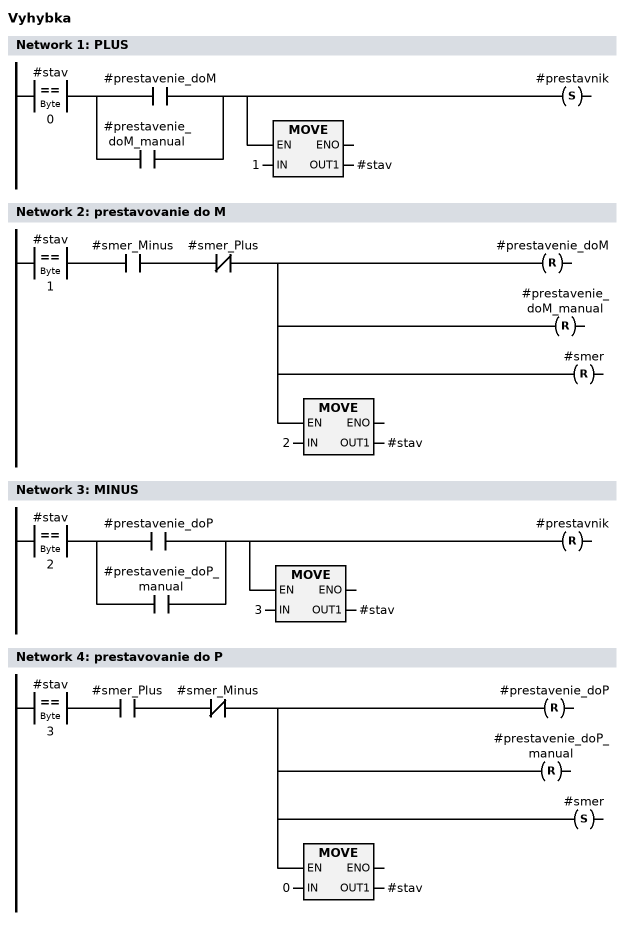
   RUNG wire#powerrail
      { S7_Templates := "SrcType := Byte" } EQ_Contact(in1 := #stav, in2 := 0)
      wire#w1
      Contact( #prestavenie_doM )
      wire#w2
      S_Coil( #prestavnik )
   END_RUNG
   RUNG wire#w1
      Contact( #prestavenie_doM_manual )
   END_RUNG wire#w2
   RUNG wire#w2
      Move(in := 1, out1 => #stav)
   END_RUNG
   // the same network as SCL:
   IF (#stav = 0) AND (#prestavenie_doM OR #prestavenie_doM_manual) THEN
       #prestavnik := TRUE;
       #stav := 1;
   END_IF;
END_REGION

REGION Network 2: prestavovanie do M
   RUNG wire#powerrail
      { S7_Templates := "SrcType := Byte" } EQ_Contact(in1 := #stav, in2 := 1)
      Contact( #smer_Minus )
      I_Contact( #smer_Plus )
      wire#w1
      R_Coil( #prestavenie_doM )
   END_RUNG
   RUNG wire#w1
      R_Coil( #prestavenie_doM_manual )
   END_RUNG
   RUNG wire#w1
      R_Coil( #smer )
   END_RUNG
   RUNG wire#w1
      Move(in := 2, out1 => #stav)
   END_RUNG
   // the same network as SCL:
   IF (#stav = 1) AND #smer_Minus AND NOT #smer_Plus THEN
       #prestavenie_doM := FALSE;
       #prestavenie_doM_manual := FALSE;
       #smer := FALSE;
       #stav := 2;
   END_IF;
END_REGION

REGION Network 3: MINUS
   RUNG wire#powerrail
      { S7_Templates := "SrcType := Byte" } EQ_Contact(in1 := #stav, in2 := 2)
      wire#w1
      Contact( #prestavenie_doP )
      wire#w2
      R_Coil( #prestavnik )
   END_RUNG
   RUNG wire#w1
      Contact( #prestavenie_doP_manual )
   END_RUNG wire#w2
   RUNG wire#w2
      Move(in := 3, out1 => #stav)
   END_RUNG
   // the same network as SCL:
   IF (#stav = 2) AND (#prestavenie_doP OR #prestavenie_doP_manual) THEN
       #prestavnik := FALSE;
       #stav := 3;
   END_IF;
END_REGION

REGION Network 4: prestavovanie do P
   RUNG wire#powerrail
      { S7_Templates := "SrcType := Byte" } EQ_Contact(in1 := #stav, in2 := 3)
      Contact( #smer_Plus )
      I_Contact( #smer_Minus )
      wire#w1
      R_Coil( #prestavenie_doP )
   END_RUNG
   RUNG wire#w1
      R_Coil( #prestavenie_doP_manual )
   END_RUNG
   RUNG wire#w1
      S_Coil( #smer )
   END_RUNG
   RUNG wire#w1
      Move(in := 0, out1 => #stav)
   END_RUNG
   // the same network as SCL:
   IF (#stav = 3) AND #smer_Plus AND NOT #smer_Minus THEN
       #prestavenie_doP := FALSE;
       #prestavenie_doP_manual := FALSE;
       #smer := TRUE;
       #stav := 0;
   END_IF;
END_REGION
END_FUNCTION_BLOCK

FUNCTION_BLOCK "Detekcia_Smeru_Jazdy"   // FB8, SCL
{ S7_Optimized_Access := 'TRUE' }
VERSION : 0.1
   VAR_INPUT
      PU_AB : Bool;   // Priblizovaci usek-smer AB
      AU : Bool;   // Anulovaci usek
      PU_BA : Bool;   // Priblizovaci usek-smer BA
   END_VAR
   VAR_OUTPUT
      S_AB : Bool;   // Smer A->B
      S_BA : Bool;   // Smer B->A
   END_VAR
   VAR
      Stav : USInt;
   END_VAR
BEGIN
   CASE #Stav OF
       0:
           #S_AB := FALSE;
           #S_BA := FALSE;

           IF ((#PU_AB) AND NOT (#AU) AND NOT (#PU_BA)) THEN
               #Stav := 1;
           END_IF;

           IF (NOT (#PU_AB) AND NOT (#AU) AND (#PU_BA)) THEN
               #Stav := 2;
           END_IF;

       1:
           #S_AB := TRUE;
           #S_BA := FALSE;

           IF (NOT (#PU_AB) AND NOT (#AU) AND NOT (#PU_BA)) THEN
               #Stav := 0;
           END_IF;

       2:
           #S_AB := FALSE;
           #S_BA := TRUE;

           IF (NOT (#PU_AB) AND NOT (#AU) AND NOT (#PU_BA)) THEN
               #Stav := 0;
           END_IF;
   END_CASE;
END_FUNCTION_BLOCK

ORGANIZATION_BLOCK "Main"   // OB1, LAD, ProgramCycle
TITLE = "Main Program Sweep (Cycle)"
{ S7_Optimized_Access := 'TRUE' }
VERSION : 0.1
   VAR_INPUT
      Initial_Call : Bool;   // Initial call of this OB
      Remanence : Bool;   // =True, if remanent data are available
   END_VAR
BEGIN

REGION Network 1: Lo/PrLo
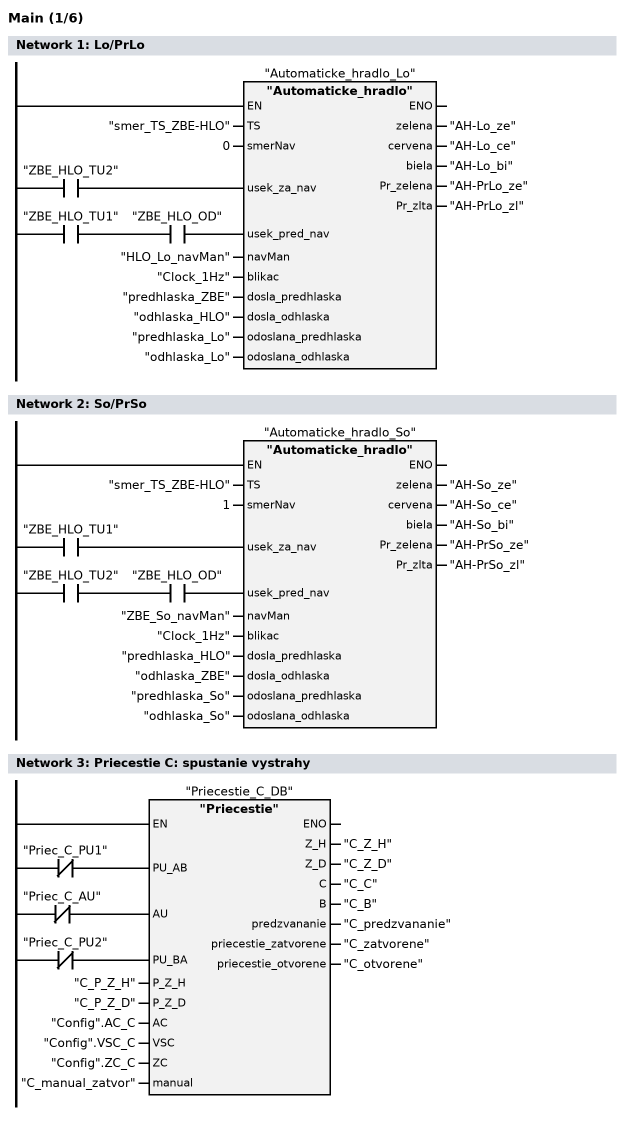
   RUNG wire#powerrail
      "Automaticke_hradlo_Lo"(usek_za_nav := wire#w1, usek_pred_nav := wire#w2, TS := "smer_TS_ZBE-HLO", smerNav := 0, navMan := "HLO_Lo_navMan", blikac := "Clock_1Hz", dosla_predhlaska := "predhlaska_ZBE", dosla_odhlaska := "odhlaska_HLO", odoslana_predhlaska := "predhlaska_Lo", odoslana_odhlaska := "odhlaska_Lo", zelena => "AH-Lo_ze", cervena => "AH-Lo_ce", biela => "AH-Lo_bi", Pr_zelena => "AH-PrLo_ze", Pr_zlta => "AH-PrLo_zl")
   END_RUNG
   RUNG wire#powerrail
      Contact( "ZBE_HLO_TU2" )
   END_RUNG wire#w1
   RUNG wire#powerrail
      Contact( "ZBE_HLO_TU1" )
      Contact( "ZBE_HLO_OD" )
   END_RUNG wire#w2
   // the same network as SCL:
   "Automaticke_hradlo_Lo"(TS := "smer_TS_ZBE-HLO",   // "Automaticke_hradlo"
                           smerNav := 0,
                           usek_za_nav := "ZBE_HLO_TU2",
                           usek_pred_nav := "ZBE_HLO_TU1" AND "ZBE_HLO_OD",
                           navMan := "HLO_Lo_navMan",
                           blikac := "Clock_1Hz",
                           dosla_predhlaska := "predhlaska_ZBE",
                           dosla_odhlaska := "odhlaska_HLO",
                           odoslana_predhlaska := "predhlaska_Lo",
                           odoslana_odhlaska := "odhlaska_Lo",
                           zelena => "AH-Lo_ze",
                           cervena => "AH-Lo_ce",
                           biela => "AH-Lo_bi",
                           Pr_zelena => "AH-PrLo_ze",
                           Pr_zlta => "AH-PrLo_zl");
END_REGION

REGION Network 2: So/PrSo
   RUNG wire#powerrail
      "Automaticke_hradlo_So"(usek_za_nav := wire#w1, usek_pred_nav := wire#w2, TS := "smer_TS_ZBE-HLO", smerNav := 1, navMan := "ZBE_So_navMan", blikac := "Clock_1Hz", dosla_predhlaska := "predhlaska_HLO", dosla_odhlaska := "odhlaska_ZBE", odoslana_predhlaska := "predhlaska_So", odoslana_odhlaska := "odhlaska_So", zelena => "AH-So_ze", cervena => "AH-So_ce", biela => "AH-So_bi", Pr_zelena => "AH-PrSo_ze", Pr_zlta => "AH-PrSo_zl")
   END_RUNG
   RUNG wire#powerrail
      Contact( "ZBE_HLO_TU1" )
   END_RUNG wire#w1
   RUNG wire#powerrail
      Contact( "ZBE_HLO_TU2" )
      Contact( "ZBE_HLO_OD" )
   END_RUNG wire#w2
   // the same network as SCL:
   "Automaticke_hradlo_So"(TS := "smer_TS_ZBE-HLO",   // "Automaticke_hradlo"
                           smerNav := 1,
                           usek_za_nav := "ZBE_HLO_TU1",
                           usek_pred_nav := "ZBE_HLO_TU2" AND "ZBE_HLO_OD",
                           navMan := "ZBE_So_navMan",
                           blikac := "Clock_1Hz",
                           dosla_predhlaska := "predhlaska_HLO",
                           dosla_odhlaska := "odhlaska_ZBE",
                           odoslana_predhlaska := "predhlaska_So",
                           odoslana_odhlaska := "odhlaska_So",
                           zelena => "AH-So_ze",
                           cervena => "AH-So_ce",
                           biela => "AH-So_bi",
                           Pr_zelena => "AH-PrSo_ze",
                           Pr_zlta => "AH-PrSo_zl");
END_REGION

REGION Network 3: Priecestie C: spustanie vystrahy
   RUNG wire#powerrail
      "Priecestie_C_DB"(PU_AB := wire#w1, AU := wire#w2, PU_BA := wire#w3, P_Z_H := "C_P_Z_H", P_Z_D := "C_P_Z_D", AC := "Config".AC_C, VSC := "Config".VSC_C, ZC := "Config".ZC_C, manual := "C_manual_zatvor", Z_H => "C_Z_H", Z_D => "C_Z_D", C => "C_C", "B" => "C_B", predzvananie => "C_predzvananie", priecestie_zatvorene => "C_zatvorene", priecestie_otvorene => "C_otvorene")
   END_RUNG
   RUNG wire#powerrail
      I_Contact( "Priec_C_PU1" )
   END_RUNG wire#w1
   RUNG wire#powerrail
      I_Contact( "Priec_C_AU" )
   END_RUNG wire#w2
   RUNG wire#powerrail
      I_Contact( "Priec_C_PU2" )
   END_RUNG wire#w3
   // the same network as SCL:
   "Priecestie_C_DB"(PU_AB := NOT "Priec_C_PU1",   // "Priecestie"
                     AU := NOT "Priec_C_AU",
                     PU_BA := NOT "Priec_C_PU2",
                     P_Z_H := "C_P_Z_H",
                     P_Z_D := "C_P_Z_D",
                     AC := "Config".AC_C,
                     VSC := "Config".VSC_C,
                     ZC := "Config".ZC_C,
                     manual := "C_manual_zatvor",
                     Z_H => "C_Z_H",
                     Z_D => "C_Z_D",
                     C => "C_C",
                     "B" => "C_B",
                     predzvananie => "C_predzvananie",
                     priecestie_zatvorene => "C_zatvorene",
                     priecestie_otvorene => "C_otvorene");
END_REGION

REGION Network 4: Priecestie E: spustanie vystrahy
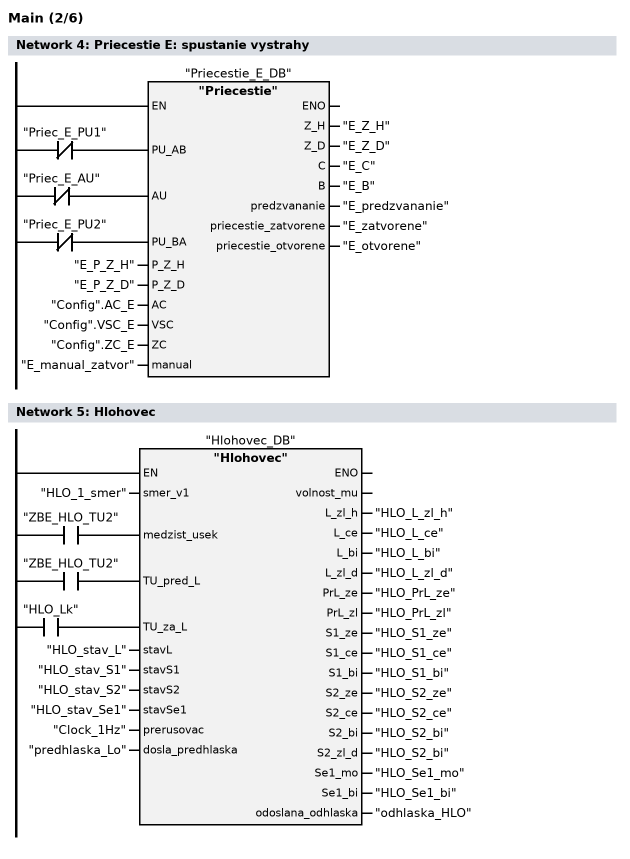
   RUNG wire#powerrail
      "Priecestie_E_DB"(PU_AB := wire#w1, AU := wire#w2, PU_BA := wire#w3, P_Z_H := "E_P_Z_H", P_Z_D := "E_P_Z_D", AC := "Config".AC_E, VSC := "Config".VSC_E, ZC := "Config".ZC_E, manual := "E_manual_zatvor", Z_H => "E_Z_H", Z_D => "E_Z_D", C => "E_C", "B" => "E_B", predzvananie => "E_predzvananie", priecestie_zatvorene => "E_zatvorene", priecestie_otvorene => "E_otvorene")
   END_RUNG
   RUNG wire#powerrail
      I_Contact( "Priec_E_PU1" )
   END_RUNG wire#w1
   RUNG wire#powerrail
      I_Contact( "Priec_E_AU" )
   END_RUNG wire#w2
   RUNG wire#powerrail
      I_Contact( "Priec_E_PU2" )
   END_RUNG wire#w3
   // the same network as SCL:
   "Priecestie_E_DB"(PU_AB := NOT "Priec_E_PU1",   // "Priecestie"
                     AU := NOT "Priec_E_AU",
                     PU_BA := NOT "Priec_E_PU2",
                     P_Z_H := "E_P_Z_H",
                     P_Z_D := "E_P_Z_D",
                     AC := "Config".AC_E,
                     VSC := "Config".VSC_E,
                     ZC := "Config".ZC_E,
                     manual := "E_manual_zatvor",
                     Z_H => "E_Z_H",
                     Z_D => "E_Z_D",
                     C => "E_C",
                     "B" => "E_B",
                     predzvananie => "E_predzvananie",
                     priecestie_zatvorene => "E_zatvorene",
                     priecestie_otvorene => "E_otvorene");
END_REGION

REGION Network 5: Hlohovec
   RUNG wire#powerrail
      "Hlohovec_DB"(medzist_usek := wire#w1, TU_pred_L := wire#w2, TU_za_L := wire#w3, smer_v1 := "HLO_1_smer", stavL := "HLO_stav_L", stavS1 := "HLO_stav_S1", stavS2 := "HLO_stav_S2", stavSe1 := "HLO_stav_Se1", prerusovac := "Clock_1Hz", dosla_predhlaska := "predhlaska_Lo", volnost_mu =>, L_zl_h => "HLO_L_zl_h", L_ce => "HLO_L_ce", L_bi => "HLO_L_bi", L_zl_d => "HLO_L_zl_d", PrL_ze => "HLO_PrL_ze", PrL_zl => "HLO_PrL_zl", S1_ze => "HLO_S1_ze", S1_ce => "HLO_S1_ce", S1_bi => "HLO_S1_bi", S2_ze => "HLO_S2_ze", S2_ce => "HLO_S2_ce", S2_bi => "HLO_S2_bi", S2_zl_d => "HLO_S2_bi", Se1_mo => "HLO_Se1_mo", Se1_bi => "HLO_Se1_bi", odoslana_odhlaska => "odhlaska_HLO")
   END_RUNG
   RUNG wire#powerrail
      Contact( "ZBE_HLO_TU2" )
   END_RUNG wire#w1
   RUNG wire#powerrail
      Contact( "ZBE_HLO_TU2" )
   END_RUNG wire#w2
   RUNG wire#powerrail
      Contact( "HLO_Lk" )
   END_RUNG wire#w3
   // the same network as SCL:
   "Hlohovec_DB"(smer_v1 := "HLO_1_smer",   // "Hlohovec"
                 medzist_usek := "ZBE_HLO_TU2",
                 TU_pred_L := "ZBE_HLO_TU2",
                 TU_za_L := "HLO_Lk",
                 stavL := "HLO_stav_L",
                 stavS1 := "HLO_stav_S1",
                 stavS2 := "HLO_stav_S2",
                 stavSe1 := "HLO_stav_Se1",
                 prerusovac := "Clock_1Hz",
                 dosla_predhlaska := "predhlaska_Lo",
                 L_zl_h => "HLO_L_zl_h",
                 L_ce => "HLO_L_ce",
                 L_bi => "HLO_L_bi",
                 L_zl_d => "HLO_L_zl_d",
                 PrL_ze => "HLO_PrL_ze",
                 PrL_zl => "HLO_PrL_zl",
                 S1_ze => "HLO_S1_ze",
                 S1_ce => "HLO_S1_ce",
                 S1_bi => "HLO_S1_bi",
                 S2_ze => "HLO_S2_ze",
                 S2_ce => "HLO_S2_ce",
                 S2_bi => "HLO_S2_bi",
                 S2_zl_d => "HLO_S2_bi",
                 Se1_mo => "HLO_Se1_mo",
                 Se1_bi => "HLO_Se1_bi",
                 odoslana_odhlaska => "odhlaska_HLO");
END_REGION

REGION Network 6: Zbehy
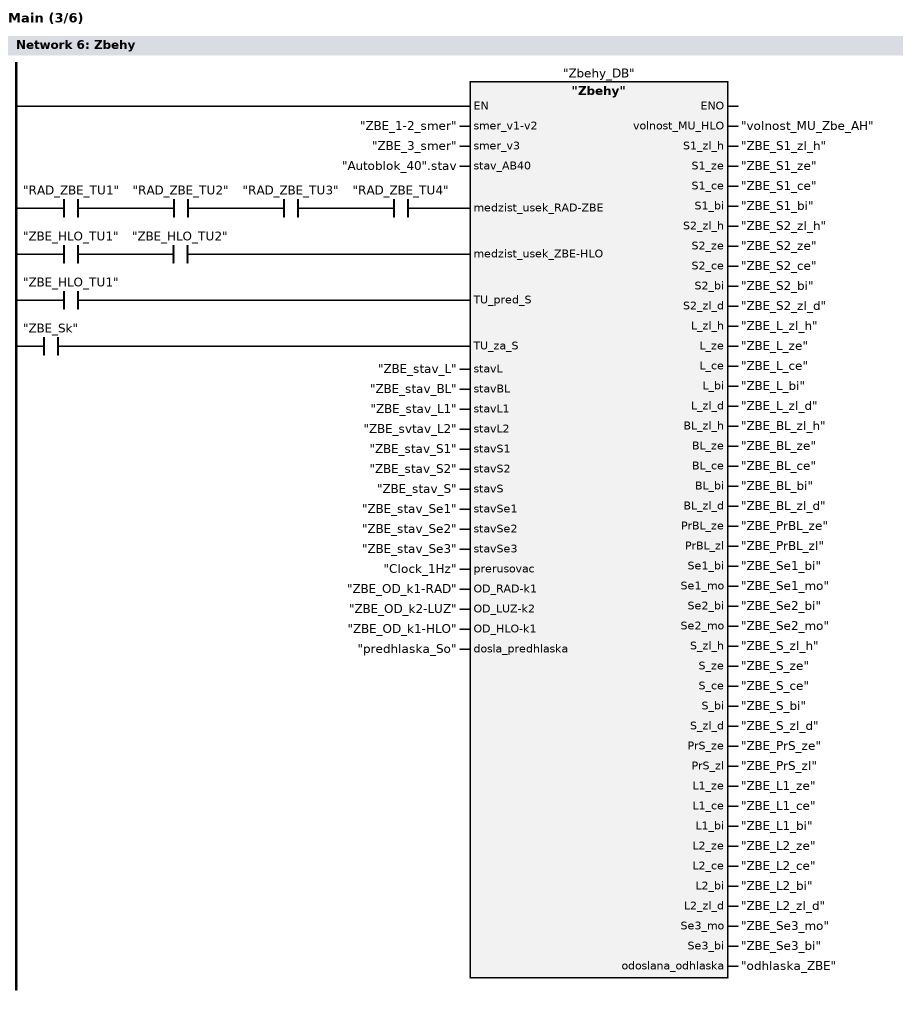
   RUNG wire#powerrail
      "Zbehy_DB"("medzist_usek_RAD-ZBE" := wire#w1, "medzist_usek_ZBE-HLO" := wire#w2, TU_pred_S := wire#w3, TU_za_S := wire#w4, "smer_v1-v2" := "ZBE_1-2_smer", smer_v3 := "ZBE_3_smer", stav_AB40 := "Autoblok_40".stav, stavL := "ZBE_stav_L", stavBL := "ZBE_stav_BL", stavL1 := "ZBE_stav_L1", stavL2 := "ZBE_svtav_L2", stavS1 := "ZBE_stav_S1", stavS2 := "ZBE_stav_S2", stavS := "ZBE_stav_S", stavSe1 := "ZBE_stav_Se1", stavSe2 := "ZBE_stav_Se2", stavSe3 := "ZBE_stav_Se3", prerusovac := "Clock_1Hz", "OD_RAD-k1" := "ZBE_OD_k1-RAD", "OD_LUZ-k2" := "ZBE_OD_k2-LUZ", "OD_HLO-k1" := "ZBE_OD_k1-HLO", dosla_predhlaska := "predhlaska_So", volnost_MU_HLO => "volnost_MU_Zbe_AH", S1_zl_h => "ZBE_S1_zl_h", S1_ze => "ZBE_S1_ze", S1_ce => "ZBE_S1_ce", S1_bi => "ZBE_S1_bi", S2_zl_h => "ZBE_S2_zl_h", S2_ze => "ZBE_S2_ze", S2_ce => "ZBE_S2_ce", S2_bi => "ZBE_S2_bi", S2_zl_d => "ZBE_S2_zl_d", L_zl_h => "ZBE_L_zl_h", L_ze => "ZBE_L_ze", L_ce => "ZBE_L_ce", L_bi => "ZBE_L_bi", L_zl_d => "ZBE_L_zl_d", BL_zl_h => "ZBE_BL_zl_h", BL_ze => "ZBE_BL_ze", BL_ce => "ZBE_BL_ce", BL_bi => "ZBE_BL_bi", BL_zl_d => "ZBE_BL_zl_d", PrBL_ze => "ZBE_PrBL_ze", PrBL_zl => "ZBE_PrBL_zl", Se1_bi => "ZBE_Se1_bi", Se1_mo => "ZBE_Se1_mo", Se2_bi => "ZBE_Se2_bi", Se2_mo => "ZBE_Se2_mo", S_zl_h => "ZBE_S_zl_h", S_ze => "ZBE_S_ze", S_ce => "ZBE_S_ce", S_bi => "ZBE_S_bi", S_zl_d => "ZBE_S_zl_d", PrS_ze => "ZBE_PrS_ze", PrS_zl => "ZBE_PrS_zl", L1_ze => "ZBE_L1_ze", L1_ce => "ZBE_L1_ce", L1_bi => "ZBE_L1_bi", L2_ze => "ZBE_L2_ze", L2_ce => "ZBE_L2_ce", L2_bi => "ZBE_L2_bi", L2_zl_d => "ZBE_L2_zl_d", Se3_mo => "ZBE_Se3_mo", Se3_bi => "ZBE_Se3_bi", odoslana_odhlaska => "odhlaska_ZBE")
   END_RUNG
   RUNG wire#powerrail
      Contact( "RAD_ZBE_TU1" )
      Contact( "RAD_ZBE_TU2" )
      Contact( "RAD_ZBE_TU3" )
      Contact( "RAD_ZBE_TU4" )
   END_RUNG wire#w1
   RUNG wire#powerrail
      Contact( "ZBE_HLO_TU1" )
      Contact( "ZBE_HLO_TU2" )
   END_RUNG wire#w2
   RUNG wire#powerrail
      Contact( "ZBE_HLO_TU1" )
   END_RUNG wire#w3
   RUNG wire#powerrail
      Contact( "ZBE_Sk" )
   END_RUNG wire#w4
   // the same network as SCL:
   "Zbehy_DB"("smer_v1-v2" := "ZBE_1-2_smer",   // "Zbehy"
              smer_v3 := "ZBE_3_smer",
              stav_AB40 := "Autoblok_40".stav,
              "medzist_usek_RAD-ZBE" := "RAD_ZBE_TU1" AND "RAD_ZBE_TU2" AND "RAD_ZBE_TU3" AND "RAD_ZBE_TU4",
              "medzist_usek_ZBE-HLO" := "ZBE_HLO_TU1" AND "ZBE_HLO_TU2",
              TU_pred_S := "ZBE_HLO_TU1",
              TU_za_S := "ZBE_Sk",
              stavL := "ZBE_stav_L",
              stavBL := "ZBE_stav_BL",
              stavL1 := "ZBE_stav_L1",
              stavL2 := "ZBE_svtav_L2",
              stavS1 := "ZBE_stav_S1",
              stavS2 := "ZBE_stav_S2",
              stavS := "ZBE_stav_S",
              stavSe1 := "ZBE_stav_Se1",
              stavSe2 := "ZBE_stav_Se2",
              stavSe3 := "ZBE_stav_Se3",
              prerusovac := "Clock_1Hz",
              "OD_RAD-k1" := "ZBE_OD_k1-RAD",
              "OD_LUZ-k2" := "ZBE_OD_k2-LUZ",
              "OD_HLO-k1" := "ZBE_OD_k1-HLO",
              dosla_predhlaska := "predhlaska_So",
              volnost_MU_HLO => "volnost_MU_Zbe_AH",
              S1_zl_h => "ZBE_S1_zl_h",
              S1_ze => "ZBE_S1_ze",
              S1_ce => "ZBE_S1_ce",
              S1_bi => "ZBE_S1_bi",
              S2_zl_h => "ZBE_S2_zl_h",
              S2_ze => "ZBE_S2_ze",
              S2_ce => "ZBE_S2_ce",
              S2_bi => "ZBE_S2_bi",
              S2_zl_d => "ZBE_S2_zl_d",
              L_zl_h => "ZBE_L_zl_h",
              L_ze => "ZBE_L_ze",
              L_ce => "ZBE_L_ce",
              L_bi => "ZBE_L_bi",
              L_zl_d => "ZBE_L_zl_d",
              BL_zl_h => "ZBE_BL_zl_h",
              BL_ze => "ZBE_BL_ze",
              BL_ce => "ZBE_BL_ce",
              BL_bi => "ZBE_BL_bi",
              BL_zl_d => "ZBE_BL_zl_d",
              PrBL_ze => "ZBE_PrBL_ze",
              PrBL_zl => "ZBE_PrBL_zl",
              Se1_bi => "ZBE_Se1_bi",
              Se1_mo => "ZBE_Se1_mo",
              Se2_bi => "ZBE_Se2_bi",
              Se2_mo => "ZBE_Se2_mo",
              S_zl_h => "ZBE_S_zl_h",
              S_ze => "ZBE_S_ze",
              S_ce => "ZBE_S_ce",
              S_bi => "ZBE_S_bi",
              S_zl_d => "ZBE_S_zl_d",
              PrS_ze => "ZBE_PrS_ze",
              PrS_zl => "ZBE_PrS_zl",
              L1_ze => "ZBE_L1_ze",
              L1_ce => "ZBE_L1_ce",
              L1_bi => "ZBE_L1_bi",
              L2_ze => "ZBE_L2_ze",
              L2_ce => "ZBE_L2_ce",
              L2_bi => "ZBE_L2_bi",
              L2_zl_d => "ZBE_L2_zl_d",
              Se3_mo => "ZBE_Se3_mo",
              Se3_bi => "ZBE_Se3_bi",
              odoslana_odhlaska => "odhlaska_ZBE");
END_REGION

REGION Network 7: Radosina
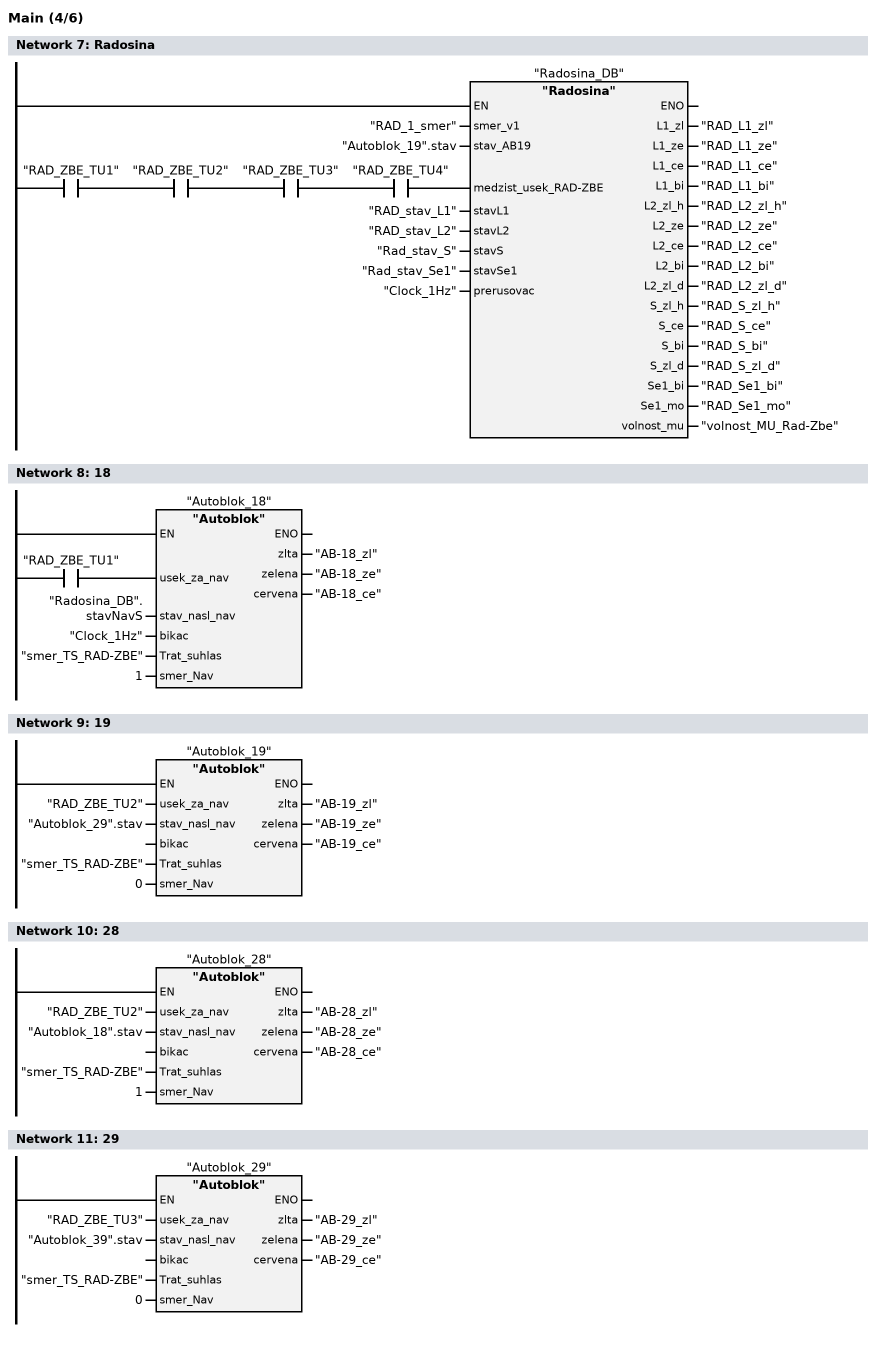
   RUNG wire#powerrail
      "Radosina_DB"("medzist_usek_RAD-ZBE" := wire#w1, smer_v1 := "RAD_1_smer", stav_AB19 := "Autoblok_19".stav, stavL1 := "RAD_stav_L1", stavL2 := "RAD_stav_L2", stavS := "Rad_stav_S", stavSe1 := "Rad_stav_Se1", prerusovac := "Clock_1Hz", L1_zl => "RAD_L1_zl", L1_ze => "RAD_L1_ze", L1_ce => "RAD_L1_ce", L1_bi => "RAD_L1_bi", L2_zl_h => "RAD_L2_zl_h", L2_ze => "RAD_L2_ze", L2_ce => "RAD_L2_ce", L2_bi => "RAD_L2_bi", L2_zl_d => "RAD_L2_zl_d", S_zl_h => "RAD_S_zl_h", S_ce => "RAD_S_ce", S_bi => "RAD_S_bi", S_zl_d => "RAD_S_zl_d", Se1_bi => "RAD_Se1_bi", Se1_mo => "RAD_Se1_mo", volnost_mu => "volnost_MU_Rad-Zbe")
   END_RUNG
   RUNG wire#powerrail
      Contact( "RAD_ZBE_TU1" )
      Contact( "RAD_ZBE_TU2" )
      Contact( "RAD_ZBE_TU3" )
      Contact( "RAD_ZBE_TU4" )
   END_RUNG wire#w1
   // the same network as SCL:
   "Radosina_DB"(smer_v1 := "RAD_1_smer",   // "Radosina"
                 stav_AB19 := "Autoblok_19".stav,
                 "medzist_usek_RAD-ZBE" := "RAD_ZBE_TU1" AND "RAD_ZBE_TU2" AND "RAD_ZBE_TU3" AND "RAD_ZBE_TU4",
                 stavL1 := "RAD_stav_L1",
                 stavL2 := "RAD_stav_L2",
                 stavS := "Rad_stav_S",
                 stavSe1 := "Rad_stav_Se1",
                 prerusovac := "Clock_1Hz",
                 L1_zl => "RAD_L1_zl",
                 L1_ze => "RAD_L1_ze",
                 L1_ce => "RAD_L1_ce",
                 L1_bi => "RAD_L1_bi",
                 L2_zl_h => "RAD_L2_zl_h",
                 L2_ze => "RAD_L2_ze",
                 L2_ce => "RAD_L2_ce",
                 L2_bi => "RAD_L2_bi",
                 L2_zl_d => "RAD_L2_zl_d",
                 S_zl_h => "RAD_S_zl_h",
                 S_ce => "RAD_S_ce",
                 S_bi => "RAD_S_bi",
                 S_zl_d => "RAD_S_zl_d",
                 Se1_bi => "RAD_Se1_bi",
                 Se1_mo => "RAD_Se1_mo",
                 volnost_mu => "volnost_MU_Rad-Zbe");
END_REGION

REGION Network 8: 18
   RUNG wire#powerrail
      "Autoblok_18"(usek_za_nav := wire#w1, stav_nasl_nav := "Radosina_DB".stavNavS, bikac := "Clock_1Hz", Trat_suhlas := "smer_TS_RAD-ZBE", smer_Nav := 1, zlta => "AB-18_zl", zelena => "AB-18_ze", cervena => "AB-18_ce")
   END_RUNG
   RUNG wire#powerrail
      Contact( "RAD_ZBE_TU1" )
   END_RUNG wire#w1
   // the same network as SCL:
   "Autoblok_18"(usek_za_nav := "RAD_ZBE_TU1",   // "Autoblok"
                 stav_nasl_nav := "Radosina_DB".stavNavS,
                 bikac := "Clock_1Hz",
                 Trat_suhlas := "smer_TS_RAD-ZBE",
                 smer_Nav := 1,
                 zlta => "AB-18_zl",
                 zelena => "AB-18_ze",
                 cervena => "AB-18_ce");
END_REGION

REGION Network 9: 19
   RUNG wire#powerrail
      "Autoblok_19"(usek_za_nav := "RAD_ZBE_TU2", stav_nasl_nav := "Autoblok_29".stav, bikac :=, Trat_suhlas := "smer_TS_RAD-ZBE", smer_Nav := 0, zlta => "AB-19_zl", zelena => "AB-19_ze", cervena => "AB-19_ce")
   END_RUNG
   // the same network as SCL:
   "Autoblok_19"(usek_za_nav := "RAD_ZBE_TU2",   // "Autoblok"
                 stav_nasl_nav := "Autoblok_29".stav,
                 Trat_suhlas := "smer_TS_RAD-ZBE",
                 smer_Nav := 0,
                 zlta => "AB-19_zl",
                 zelena => "AB-19_ze",
                 cervena => "AB-19_ce");
END_REGION

REGION Network 10: 28
   RUNG wire#powerrail
      "Autoblok_28"(usek_za_nav := "RAD_ZBE_TU2", stav_nasl_nav := "Autoblok_18".stav, bikac :=, Trat_suhlas := "smer_TS_RAD-ZBE", smer_Nav := 1, zlta => "AB-28_zl", zelena => "AB-28_ze", cervena => "AB-28_ce")
   END_RUNG
   // the same network as SCL:
   "Autoblok_28"(usek_za_nav := "RAD_ZBE_TU2",   // "Autoblok"
                 stav_nasl_nav := "Autoblok_18".stav,
                 Trat_suhlas := "smer_TS_RAD-ZBE",
                 smer_Nav := 1,
                 zlta => "AB-28_zl",
                 zelena => "AB-28_ze",
                 cervena => "AB-28_ce");
END_REGION

REGION Network 11: 29
   RUNG wire#powerrail
      "Autoblok_29"(usek_za_nav := "RAD_ZBE_TU3", stav_nasl_nav := "Autoblok_39".stav, bikac :=, Trat_suhlas := "smer_TS_RAD-ZBE", smer_Nav := 0, zlta => "AB-29_zl", zelena => "AB-29_ze", cervena => "AB-29_ce")
   END_RUNG
   // the same network as SCL:
   "Autoblok_29"(usek_za_nav := "RAD_ZBE_TU3",   // "Autoblok"
                 stav_nasl_nav := "Autoblok_39".stav,
                 Trat_suhlas := "smer_TS_RAD-ZBE",
                 smer_Nav := 0,
                 zlta => "AB-29_zl",
                 zelena => "AB-29_ze",
                 cervena => "AB-29_ce");
END_REGION

REGION Network 12: 40
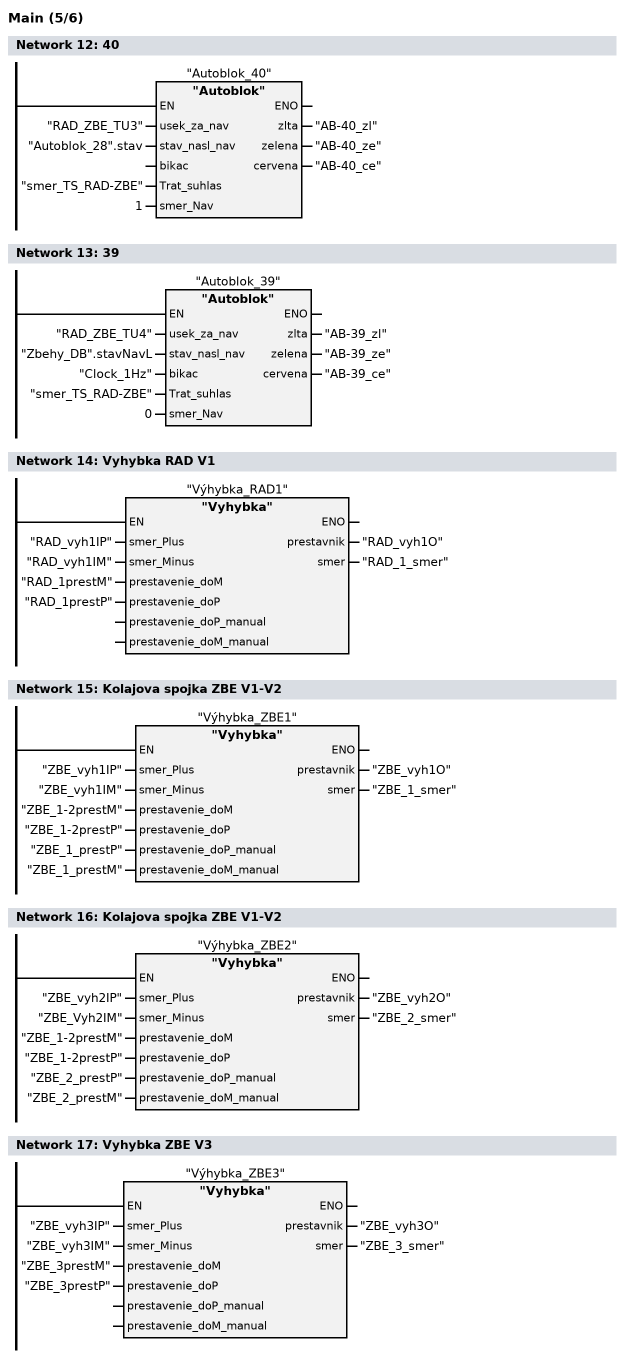
   RUNG wire#powerrail
      "Autoblok_40"(usek_za_nav := "RAD_ZBE_TU3", stav_nasl_nav := "Autoblok_28".stav, bikac :=, Trat_suhlas := "smer_TS_RAD-ZBE", smer_Nav := 1, zlta => "AB-40_zl", zelena => "AB-40_ze", cervena => "AB-40_ce")
   END_RUNG
   // the same network as SCL:
   "Autoblok_40"(usek_za_nav := "RAD_ZBE_TU3",   // "Autoblok"
                 stav_nasl_nav := "Autoblok_28".stav,
                 Trat_suhlas := "smer_TS_RAD-ZBE",
                 smer_Nav := 1,
                 zlta => "AB-40_zl",
                 zelena => "AB-40_ze",
                 cervena => "AB-40_ce");
END_REGION

REGION Network 13: 39
   RUNG wire#powerrail
      "Autoblok_39"(usek_za_nav := "RAD_ZBE_TU4", stav_nasl_nav := "Zbehy_DB".stavNavL, bikac := "Clock_1Hz", Trat_suhlas := "smer_TS_RAD-ZBE", smer_Nav := 0, zlta => "AB-39_zl", zelena => "AB-39_ze", cervena => "AB-39_ce")
   END_RUNG
   // the same network as SCL:
   "Autoblok_39"(usek_za_nav := "RAD_ZBE_TU4",   // "Autoblok"
                 stav_nasl_nav := "Zbehy_DB".stavNavL,
                 bikac := "Clock_1Hz",
                 Trat_suhlas := "smer_TS_RAD-ZBE",
                 smer_Nav := 0,
                 zlta => "AB-39_zl",
                 zelena => "AB-39_ze",
                 cervena => "AB-39_ce");
END_REGION

REGION Network 14: Vyhybka RAD V1
   RUNG wire#powerrail
      "Výhybka_RAD1"(smer_Plus := "RAD_vyh1IP", smer_Minus := "RAD_vyh1IM", prestavenie_doM := "RAD_1prestM", prestavenie_doP := "RAD_1prestP", prestavenie_doP_manual :=, prestavenie_doM_manual :=, prestavnik => "RAD_vyh1O", smer => "RAD_1_smer")
   END_RUNG
   // the same network as SCL:
   "Výhybka_RAD1"(smer_Plus := "RAD_vyh1IP",   // "Vyhybka"
                  smer_Minus := "RAD_vyh1IM",
                  prestavenie_doM := "RAD_1prestM",
                  prestavenie_doP := "RAD_1prestP",
                  prestavnik => "RAD_vyh1O",
                  smer => "RAD_1_smer");
END_REGION

REGION Network 15: Kolajova spojka ZBE V1-V2
   RUNG wire#powerrail
      "Výhybka_ZBE1"(smer_Plus := "ZBE_vyh1IP", smer_Minus := "ZBE_vyh1IM", prestavenie_doM := "ZBE_1-2prestM", prestavenie_doP := "ZBE_1-2prestP", prestavenie_doP_manual := "ZBE_1_prestP", prestavenie_doM_manual := "ZBE_1_prestM", prestavnik => "ZBE_vyh1O", smer => "ZBE_1_smer")
   END_RUNG
   // the same network as SCL:
   "Výhybka_ZBE1"(smer_Plus := "ZBE_vyh1IP",   // "Vyhybka"
                  smer_Minus := "ZBE_vyh1IM",
                  prestavenie_doM := "ZBE_1-2prestM",
                  prestavenie_doP := "ZBE_1-2prestP",
                  prestavenie_doP_manual := "ZBE_1_prestP",
                  prestavenie_doM_manual := "ZBE_1_prestM",
                  prestavnik => "ZBE_vyh1O",
                  smer => "ZBE_1_smer");
END_REGION

REGION Network 16: Kolajova spojka ZBE V1-V2
   RUNG wire#powerrail
      "Výhybka_ZBE2"(smer_Plus := "ZBE_vyh2IP", smer_Minus := "ZBE_Vyh2IM", prestavenie_doM := "ZBE_1-2prestM", prestavenie_doP := "ZBE_1-2prestP", prestavenie_doP_manual := "ZBE_2_prestP", prestavenie_doM_manual := "ZBE_2_prestM", prestavnik => "ZBE_vyh2O", smer => "ZBE_2_smer")
   END_RUNG
   // the same network as SCL:
   "Výhybka_ZBE2"(smer_Plus := "ZBE_vyh2IP",   // "Vyhybka"
                  smer_Minus := "ZBE_Vyh2IM",
                  prestavenie_doM := "ZBE_1-2prestM",
                  prestavenie_doP := "ZBE_1-2prestP",
                  prestavenie_doP_manual := "ZBE_2_prestP",
                  prestavenie_doM_manual := "ZBE_2_prestM",
                  prestavnik => "ZBE_vyh2O",
                  smer => "ZBE_2_smer");
END_REGION

REGION Network 17: Vyhybka ZBE V3
   RUNG wire#powerrail
      "Výhybka_ZBE3"(smer_Plus := "ZBE_vyh3IP", smer_Minus := "ZBE_vyh3IM", prestavenie_doM := "ZBE_3prestM", prestavenie_doP := "ZBE_3prestP", prestavenie_doP_manual :=, prestavenie_doM_manual :=, prestavnik => "ZBE_vyh3O", smer => "ZBE_3_smer")
   END_RUNG
   // the same network as SCL:
   "Výhybka_ZBE3"(smer_Plus := "ZBE_vyh3IP",   // "Vyhybka"
                  smer_Minus := "ZBE_vyh3IM",
                  prestavenie_doM := "ZBE_3prestM",
                  prestavenie_doP := "ZBE_3prestP",
                  prestavnik => "ZBE_vyh3O",
                  smer => "ZBE_3_smer");
END_REGION

REGION Network 18: Vyhybka HLO V1
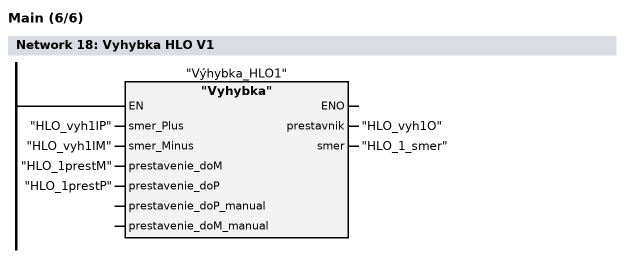
   RUNG wire#powerrail
      "Výhybka_HLO1"(smer_Plus := "HLO_vyh1IP", smer_Minus := "HLO_vyh1IM", prestavenie_doM := "HLO_1prestM", prestavenie_doP := "HLO_1prestP", prestavenie_doP_manual :=, prestavenie_doM_manual :=, prestavnik => "HLO_vyh1O", smer => "HLO_1_smer")
   END_RUNG
   // the same network as SCL:
   "Výhybka_HLO1"(smer_Plus := "HLO_vyh1IP",   // "Vyhybka"
                  smer_Minus := "HLO_vyh1IM",
                  prestavenie_doM := "HLO_1prestM",
                  prestavenie_doP := "HLO_1prestP",
                  prestavnik => "HLO_vyh1O",
                  smer => "HLO_1_smer");
END_REGION
END_ORGANIZATION_BLOCK